{attribute 'linkalways'} 
{attribute 'no_explicit_call' := 'This FB is a CLASS and must be accessed using methods or properties'}
{attribute 'enable_dynamic_creation'}
FUNCTION_BLOCK _Array0to3OfREAL EXTENDS ArrayDatatypeBase_1D
VAR CONSTANT
	lBound : DINT := 0;
	uBound : DINT := 3;
END_VAR
VAR
	localData : ARRAY [lBound..uBound] OF REAL;
	activeData : REFERENCE TO ARRAY [lBound..uBound] OF REAL REF= localData;
	elements : ARRAY [lBound..uBound] OF _REAL(0.0);
	baseType : _REAL(0.0);
END_VAR

PROPERTY PUBLIC Address : PVOID
GET
Address := ADR(activeData);
END_GET
END_PROPERTY

PROPERTY PUBLIC BaseDatatype : I_Datatype
GET
BaseDatatype := baseType;
END_GET
END_PROPERTY

METHOD PUBLIC ClearReference
VAR_INPUT
END_VAR
activeData REF= localData;
SetElementReference();
END_METHOD

METHOD PUBLIC Clone : I_Datatype
VAR
    pClone : POINTER TO _Array0to3OfREAL;
END_VAR
pClone := __NEW(_Array0to3OfREAL());
pClone^.Value := Value;
Clone := pClone^;
END_METHOD

METHOD FB_init : BOOL
VAR_INPUT
	bInitRetains : BOOL; // if TRUE, the retain variables are initialized (warm start / cold start)
	bInCopyCode : BOOL;  // if TRUE, the instance afterwards gets moved into the copy code (online change)
END_VAR
SetElementReference();
END_METHOD

METHOD PUBLIC MakeReferenceTo
VAR_INPUT
	ReferenceTarget : REFERENCE TO ARRAY [lBound..uBound] OF REAL;
END_VAR
activeData REF= ReferenceTarget;
SetElementReference();
END_METHOD

METHOD PROTECTED OnSerializeArrayValues
VAR_INPUT
	Serializer : I_Serializer;
END_VAR
VAR
	i : DINT;
END_VAR
FOR i := lBound TO uBound DO
	elements[i].SerializeWith(Serializer);
END_FOR
END_METHOD

METHOD PROTECTED SetElementReference
VAR_INPUT
END_VAR
VAR
	i : DINT;
END_VAR
FOR i := lBound TO uBound DO
	elements[i].MakeReferenceTo(activeData[i]);
END_FOR
END_METHOD

PROPERTY PUBLIC Size : UDINT
GET
Size := SIZEOF(activeData);
END_GET
END_PROPERTY

METHOD PROTECTED TryDeserializeArrayValues : BOOL
VAR_INPUT
	Deserializer : I_Deserializer;
	Feedback : I_DeserializerFeedback;
END_VAR
VAR
	enumerator : I_DeserializerArrayForwardEnumerator;
	i : DINT;
END_VAR
enumerator := Deserializer.GetArrayEnumerator();
i := lBound;

WHILE enumerator.MoveNext() AND i <= uBound DO
	
	IF NOT elements[i].TryDeserializeFrom(enumerator.Current, Feedback) THEN
		EXIT;
	END_IF
	i := i + 1;

END_WHILE
enumerator.Dispose();
END_METHOD

METHOD PUBLIC TryGetElementAsDatatypeByIndex : BOOL
VAR_INPUT
	Index : DINT;
	Destination : REFERENCE TO I_Datatype;
END_VAR
IF Index < lbound OR Index > ubound THEN
	RETURN;
END_IF

Destination := elements[Index];
TryGetElementAsDatatypeByIndex := TRUE;
END_METHOD

METHOD PUBLIC TryGetLowerBound : BOOL
VAR_INPUT
	Dimention : UDINT;
	Destination : REFERENCE TO DINT;
END_VAR
IF Dimention = 1 THEN
	Destination := lBound;
	TryGetLowerBound := TRUE;
END_IF
END_METHOD

METHOD PUBLIC TryGetUpperBound : BOOL
VAR_INPUT
	Dimention : UDINT;
	Destination : REFERENCE TO DINT;
END_VAR
IF Dimention = 1 THEN
	Destination := uBound;
	TryGetUpperBound := TRUE;
END_IF
END_METHOD

METHOD TryMakeReferenceTo : BOOL
VAR_INPUT
	Target : I_Datatype;
END_VAR
VAR
	pTargetData : POINTER TO ARRAY [lBound..uBound] OF REAL;
END_VAR
IF NOT IsEquivalentTo(Target) THEN
	RETURN;
END_IF

pTargetData := Target.Address;
activeData REF= pTargetData^;
SetElementReference();
TryMakeReferenceTo := TRUE;
END_METHOD

PROPERTY PUBLIC Value : REFERENCE TO ARRAY [lBound..uBound] OF REAL;
GET
Value ref= activeData;
END_GET
END_PROPERTY

END_FUNCTION_BLOCK

(* stored: Version 1.1.0.1, ProductVersion 3.1.4024.13
   POU _Array0to3OfREAL: Id {0fbe6eca-03f1-05cf-248a-c7d81174c9c7}, SpecialFunc None
   Folder Core: Id {78c574bf-9173-0475-1702-7265d22184f5}
   Folder Constructor: Id {da9aa09b-1ac6-0f0d-2ac2-e65f502e3857}
   Folder Protected: Id {2e978d3d-7c82-0bc8-2bbc-d92b662c14b7}
   Folder Customize: Id {270f1e24-1995-0e4a-1a60-326c5518056b}
   Property Address: Id {1030e20d-8d6e-0636-1a4f-47a2ba9dd594}
   Get Get: Id {89e8184f-e563-0df2-15f6-9aa9c825c06f}
   Property BaseDatatype: Id {f967f37e-3d8e-0f5f-1932-2169baad670c}
   Get Get: Id {bdbc9a79-4a81-03ab-116e-3faa37da7663}
   Method ClearReference: Id {1e23be15-89c2-0b85-3451-87e3742a1582}
   Method Clone: Id {277263d8-e3f2-0110-0c99-761c13433555}
   Method FB_init: Id {ee991391-74dd-05a2-275d-b338b19d9f4d}
   Method MakeReferenceTo: Id {bc0496ec-ec04-0065-150a-d7995cc50fdb}
   Method OnSerializeArrayValues: Id {2aacf54f-afaa-0022-1b96-0c4f05166108}
   Method SetElementReference: Id {3cc92e35-e784-0779-094d-a6b7f44c2ec8}
   Property Size: Id {d05707d3-7b56-0c1e-2dde-817ea2a351f3}
   Get Get: Id {e95516e5-1947-00c4-2395-b7eebb1f04ae}
   Method TryDeserializeArrayValues: Id {ee3137d1-a3c0-03c2-2639-2f76178722de}
   Method TryGetElementAsDatatypeByIndex: Id {c1530ca9-3a55-0184-01b5-c8458cc6bec0}
   Method TryGetLowerBound: Id {bd2e5ee9-0f62-0536-0033-bbe1a3864d82}
   Method TryGetUpperBound: Id {e114b3e5-7aa6-0fdd-2865-21cccfa84750}
   Method TryMakeReferenceTo: Id {0c7a0b0d-54bc-0ec0-1ca3-82bf26331b5c}
   Property Value: Id {6456918f-3f04-097a-0c1b-ac007924baaa}
   Get Get: Id {be163b59-bfa4-0bcf-1f15-a725cf22c168} *)
